FUNCTION_BLOCK FT_DERIV_10 (* Derivative with variable window size (0..9 periods) *)
  (* Standard: 61499-1 *)
  (* Version 1.0, 2025-12-21, CodingAssistant, initial API and implementation and/or initial documentation *)
  PACKAGE OSCAT::Basic::POUs::Engineering::Control;
  IMPORT OSCAT::Basic::POUs::Engineering::measurements::T_PLC_US;
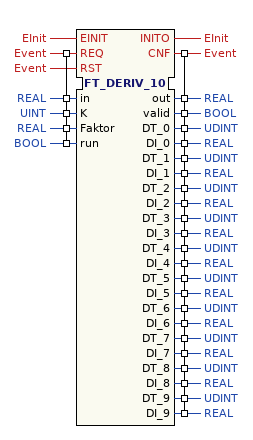
  EVENT_INPUT
    EINIT : EInit; (* Init Request *)
    REQ WITH in, K, Faktor, run; (* Normal Execution Request *)
    RST; (* Reset Buffer *)
  END_EVENT
  EVENT_OUTPUT
    INITO : EInit; (* Init Confirmation *)
    CNF WITH out, valid, DT_0, DI_0, DT_1, DI_1, DT_2, DI_2, DT_3, DI_3, DT_4, DI_4, DT_5, DI_5, DT_6, DI_6, DT_7, DI_7, DT_8, DI_8, DT_9, DI_9; (* Execution Confirmation *)
  END_EVENT
  VAR_INPUT
    in : REAL; (* Input Signal *)
    K : UINT := 0; (* Window Select: 0=1 Period, 9=10 Periods *)
    Faktor : REAL := 1.0; (* Multiplication Factor (formerly K) *)
    run : BOOL := 1; (* Enable calculation *)
  END_VAR
  VAR_OUTPUT
    out : REAL; (* Resulting Derivative based on K *)
    valid : BOOL; (* True if buffer has enough data for K *)
    DT_0 : UDINT; (* Delta T over 1 period *)
    DI_0 : REAL; (* Delta In over 1 period *)
    DT_1 : UDINT; (* Delta T over 2 period *)
    DI_1 : REAL; (* Delta In over 2 period *)
    DT_2 : UDINT; (* Delta T over 3 period *)
    DI_2 : REAL; (* Delta In over 3 period *)
    DT_3 : UDINT; (* Delta T over 4 period *)
    DI_3 : REAL; (* Delta In over 4 period *)
    DT_4 : UDINT; (* Delta T over 5 period *)
    DI_4 : REAL; (* Delta In over 5 period *)
    DT_5 : UDINT; (* Delta T over 6 period *)
    DI_5 : REAL; (* Delta In over 6 period *)
    DT_6 : UDINT; (* Delta T over 7 period *)
    DI_6 : REAL; (* Delta In over 7 period *)
    DT_7 : UDINT; (* Delta T over 8 period *)
    DI_7 : REAL; (* Delta In over 8 period *)
    DT_8 : UDINT; (* Delta T over 9 period *)
    DI_8 : REAL; (* Delta In over 9 period *)
    DT_9 : UDINT; (* Delta T over 10 period *)
    DI_9 : REAL; (* Delta In over 10 period *)
  END_VAR
  VAR CONSTANT
    MIN_PTR : INT := 0; (* ptr min *)
    MAX_PTR : INT := 10; (* ptr max *)
    MAX_CNT : INT := 11; (* cnt max *)
    INCR : INT := 1; (* increment *)
  END_VAR
  VAR
    buf_in : ARRAY [0..10] OF REAL; (* Ringbuffer Input *)
    buf_tx : ARRAY [0..10] OF UDINT; (* Ringbuffer Time *)
    ptr : INT := 0; (* Pointer to current newest *)
    cnt : INT := 0; (* Count of valid samples *)
    init_done : BOOL := FALSE;
    tx_now : UDINT;
    idx_old : INT;
    temp_dt : UDINT;
    temp_di : REAL;
  END_VAR
  EC_STATES
    EINIT : EINIT -> INITO;
    REQ : REQ -> CNF;
    RST : RST -> CNF;
  END_STATES
  ALGORITHM EINIT IN ST:
init_done := FALSE;
cnt := 0;
ptr := 0;
out := 0.0;
  END_ALGORITHM
  ALGORITHM RST IN ST:
init_done := FALSE;
cnt := 0;
ptr := 0;
out := 0.0;
valid := FALSE;
(* Arrays leeren ist in ST oft optional, hier setzen wir Zähler zurück *)
  END_ALGORITHM
  ALGORITHM REQ IN ST:
VAR_TEMP
	i : INT := 0;
END_VAR

(* 1. Initialisierung beim allerersten Durchlauf *)
IF NOT init_done THEN
	(* Erster Zyklus: Nur aktuellen Wert speichern, noch keine Berechnung möglich *)
	tx_now := T_PLC_US();
	buf_in[0] := in;
	buf_tx[0] := tx_now;

	ptr := 0;
	cnt := 1; (* Wir haben 1 gültigen Wert *)
	init_done := TRUE;

	out := 0.0;
	valid := FALSE;
	RETURN; (* Abbruch, da wir noch keine Differenz bilden können *)
END_IF;

IF run THEN
	(* 2. Neuen Wert in Ring-Buffer schreiben *)
	tx_now := T_PLC_US();

	(* Zeiger erhöhen (Ring: 0..10) *)
	ptr := ptr + INCR;
	IF ptr > MAX_PTR THEN
		ptr := MIN_PTR;
	END_IF;

	(* Werte speichern *)
	buf_in[ptr] := in;
	buf_tx[ptr] := tx_now;

	(* Gültige Samples hochzählen (Sättigung bei 11) *)
	IF cnt < MAX_CNT THEN
		cnt := cnt + INCR;
	END_IF;

	(* 3. Alle 10 Deltas berechnen und auf Ausgänge schreiben *)
	(* Hinweis: Wir machen das explizit, damit alle Pins befüllt werden *)
	(* Lokale Hilfsfunktion zur Indexberechnung: (ptr - steps + 11) MOD 11 *)
	(* Da MOD in ST manchmal negativ sein kann bei (ptr - steps), addieren wir erst 11 *)
	(* Berechnung Loop *)
	FOR i := 0 TO 9 DO
		(* Wir wollen i+1 Schritte zurückschauen. i=0 -> 1 Schritt zurück *)
		idx_old := ptr - (i + 1);
		IF idx_old < 0 THEN
			idx_old := idx_old + 11;
		END_IF;

		IF cnt > (i + 1) THEN
			(* Zeitdifferenz (UDINT Überlauf ist hier automatisch sicher) *)
			temp_dt := buf_tx[ptr] - buf_tx[idx_old];
			temp_di := buf_in[ptr] - buf_in[idx_old];
		ELSE
			temp_dt := 0;
			temp_di := 0.0;
		END_IF;

		(* Zuweisung an die expliziten Ausgänge *)
		CASE i OF
			0 :
				DT_0 := temp_dt;
				DI_0 := temp_di;
			1 :
				DT_1 := temp_dt;
				DI_1 := temp_di;
			2 :
				DT_2 := temp_dt;
				DI_2 := temp_di;
			3 :
				DT_3 := temp_dt;
				DI_3 := temp_di;
			4 :
				DT_4 := temp_dt;
				DI_4 := temp_di;
			5 :
				DT_5 := temp_dt;
				DI_5 := temp_di;
			6 :
				DT_6 := temp_dt;
				DI_6 := temp_di;
			7 :
				DT_7 := temp_dt;
				DI_7 := temp_di;
			8 :
				DT_8 := temp_dt;
				DI_8 := temp_di;
			9 :
				DT_9 := temp_dt;
				DI_9 := temp_di;
		END_CASE;
	END_FOR;

	(* 4. Hauptausgang 'out' basierend auf Eingang 'K' berechnen *)
	(* K=0 -> Wir nehmen DT_0 (1 Periode), K=9 -> DT_9 *)
	IF K > 9 THEN
		(* Fallback falls K ungültig hoch ist *)
		valid := FALSE;
		out := 0.0;
	ELSIF cnt > (UINT_TO_INT(K) + 1) THEN
		(* Wir haben genug Historie für die angeforderte Tiefe K *)
		valid := TRUE;

			(* Werte holen (über Switch/Case oder Arrayzugriff auf die Ausgänge ist in ST schwer,
			 * daher berechnen wir den Index für 'K' noch einmal kurz) *)
		idx_old := ptr - (UINT_TO_INT(K) + 1);
		IF idx_old < 0 THEN
			idx_old := idx_old + 11;
		END_IF;

		temp_dt := buf_tx[ptr] - buf_tx[idx_old];
		temp_di := buf_in[ptr] - buf_in[idx_old];

		IF temp_dt > 0 THEN
			(* Skalierung: (Delta In / Delta T µs) * 1.000.000 * Faktor *)
			out := (temp_di * 1000000.0) / UDINT_TO_REAL(temp_dt) * Faktor;
		ELSE
			out := 0.0;
		END_IF;
	ELSE
		(* Puffer noch nicht voll genug für K *)
		valid := FALSE;
		out := 0.0;
	END_IF;

ELSE
	out := 0.0;
END_IF;
  END_ALGORITHM
END_FUNCTION_BLOCK
